FUNCTION_BLOCK FB_JetNozzle1
VAR_INPUT
END_VAR
VAR_OUTPUT
END_VAR
VAR
	//Properties
	bError 					: BOOL := FALSE;
	fAngleActual 			: REAL;
	fAngleSetpoint 			: REAL := 50;
	//Raw values
	nAngleActual AT %I*		: INT;
	nAngleSetpoint AT %Q* 	: INT;
END_VAR

PROPERTY AngleActual : REAL
GET
AngleActual := THIS^.fAngleActual;
END_GET
SET
THIS^.fAngleActual := AngleActual;
END_SET
END_PROPERTY

PROPERTY AngleSetpoint : REAL
GET
AngleSetpoint := THIS^.fAngleSetpoint;
END_GET
SET
THIS^.fAngleSetpoint := AngleSetpoint;
END_SET
END_PROPERTY

PROPERTY Error : BOOL
GET
Error := THIS^.bError;
END_GET
SET
THIS^.bError := Error;
END_SET
END_PROPERTY

METHOD Run
VAR_INPUT
END_VAR
//Read feedback for opening position
fAngleActual := FC_Current4_20Raw_TO_Percentage(nAngleActual);

//Write setpoint for opening position
nAngleSetpoint := FC_Percentage_TO_Current4_20Raw(fAngleSetpoint);
END_METHOD

END_FUNCTION_BLOCK

(* stored: Version 1.1.0.1, ProductVersion 3.1.4024.0
   POU FB_JetNozzle1: Id {862fa7a9-cbec-4299-83c4-7f6af978ffb1}, SpecialFunc None
   Property AngleActual: Id {03a6d335-b321-4b7c-a46c-bec7b6f2d346}
   Get Get: Id {7c731345-d3b1-4a42-b59d-c14414f8e6e0}
   Set Set: Id {60783d93-6e7d-4586-afe1-7820ec087a08}
   Property AngleSetpoint: Id {2126b226-ab41-4520-9fc7-fdf13ffbbf04}
   Get Get: Id {fb997e4c-13d8-46e7-ba92-1345e037f2aa}
   Set Set: Id {4b5a7507-004c-4a89-a5b3-0ba15a82210d}
   Property Error: Id {6ee6b375-04ed-42a6-be6e-984d20cf10d8}
   Get Get: Id {6b22733d-b5b7-4d13-a20c-38c13b09c9ce}
   Set Set: Id {35930d66-9f27-490c-ba83-18197435a575}
   Method Run: Id {c2d807a0-0606-41c2-9945-9f2c7fb6c00d} *)
